// TIA Portal V20 program export: 0 tag tables, 0 data types, 1 data blocks, 5 code blocks (in call order from the OBs), 2 instance data blocks

DATA_BLOCK "DB_Config"   // DB3
TITLE = DB_Config
{ S7_Optimized_Access := 'TRUE' }
AUTHOR : Gemini
// stored: MemoryReserve 100
   VAR
      MaxMotors : Int;
      CycleTime : Real;
      PlantName : String;
   END_VAR
BEGIN
END_DATA_BLOCK

ORGANIZATION_BLOCK "Main"   // OB1, LAD, ProgramCycle
TITLE = "Main Program Sweep (Cycle)"
{ S7_Optimized_Access := 'TRUE' }
// stored: SetENOAutomatically false
   VAR_INPUT
      Initial_Call : Bool;   // Initial call of this OB
      Remanence : Bool;   // =True, if remanent data are available
   END_VAR
BEGIN
END_ORGANIZATION_BLOCK

FUNCTION_BLOCK "FB_MotorControl"   // FB1, SCL
{ S7_Optimized_Access := 'TRUE' }
VERSION : 0.2
// stored: MemoryReserve 100, SetENOAutomatically false
   VAR_INPUT
      bStart : Bool;
      bStop : Bool;
      bAutoStop : Bool;
   END_VAR
   VAR_OUTPUT
      bRunning : Bool;
      bFault : Bool;
   END_VAR
   VAR
      tRunTime : Time;
   END_VAR
BEGIN

   IF #bStart AND NOT #bStop AND NOT #bAutoStop THEN
       #bRunning := TRUE;
   END_IF;

   IF #bStop OR #bAutoStop THEN
       #bRunning := FALSE;
   END_IF;
END_FUNCTION_BLOCK

FUNCTION_BLOCK "FB_ValveControl"   // FB2, SCL
{ S7_Optimized_Access := 'TRUE' }
// stored: MemoryReserve 100, SetENOAutomatically false
   VAR_INPUT
      bOpen : Bool;
      bClose : Bool;
   END_VAR
   VAR_OUTPUT
      bOpened : Bool;
      bClosed : Bool;
      bFault : Bool;
   END_VAR
BEGIN

   IF #bOpen THEN
       #bOpened := TRUE;
       #bClosed := FALSE;
   END_IF;

   IF #bClose THEN
       #bOpened := FALSE;
       #bClosed := TRUE;
   END_IF;
END_FUNCTION_BLOCK

FUNCTION "FC_Diagnostic" : Void   // FC2, SCL
{ S7_Optimized_Access := 'TRUE' }
// stored: SetENOAutomatically false
   VAR_INPUT
      bFault1 : Bool;
      bFault2 : Bool;
   END_VAR
   VAR_OUTPUT
      wAlarmWord : Word;
   END_VAR
BEGIN

   #wAlarmWord.%X0 := #bFault1;
   #wAlarmWord.%X1 := #bFault2;
END_FUNCTION

FUNCTION "FC_Utilities" : Void   // FC1, SCL
{ S7_Optimized_Access := 'TRUE' }
// stored: SetENOAutomatically false
   VAR_INPUT
      rInput : Real;
      rMin : Real;
      rMax : Real;
   END_VAR
   VAR_OUTPUT
      rResult : Real;
   END_VAR
BEGIN

   #rResult := (#rInput * (#rMax - #rMin)) + #rMin;
END_FUNCTION

DATA_BLOCK "DB_Motor1"   // DB1
TITLE = DB_Motor1
AUTHOR : Gemini
// stored: InstanceOfName FB_MotorControl, InstanceOfType FB
"FB_MotorControl"
BEGIN
END_DATA_BLOCK

DATA_BLOCK "DB_Valve1"   // DB2
TITLE = DB_Valve1
AUTHOR : Gemini
// stored: InstanceOfName FB_ValveControl, InstanceOfType FB
"FB_ValveControl"
BEGIN
END_DATA_BLOCK
